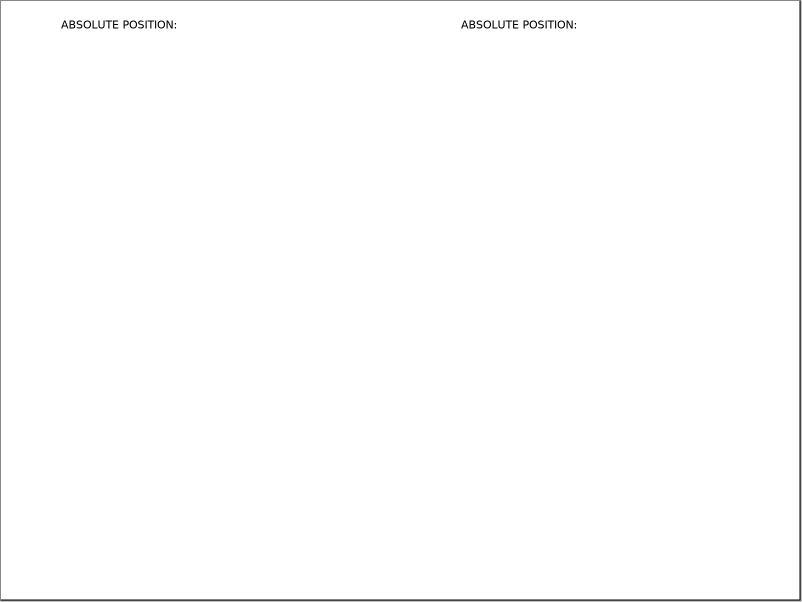
VISUALIZATION F40_Gear_In  // 802x602
    Rectangle (0,0 800x600)
    Label (10,10 170x30), "ABSOLUTE POSITION:"
    Label (410,10 170x30), "ABSOLUTE POSITION:"
END_VISUALIZATION

(* stored: Version 1.1.0.1, ProductVersion 3.1.4022.7
   Visu F40_Gear_In: Id {d2bf7a0b-7311-41f4-8a2c-33759a156bb9} *)
